SYSTEM TEST_BUTTON_LGHT (* System Configuration *)
  (* Standard: 61499-1 *)
  (* Version 0.3, 2003-12-05, JHC, Rockwell Automation, Renamed from NEWSYSTEM. *)
  (* Version 0.2, 2002-11-05, JHC, Rockwell Automation, Fixed missing (empty) FBD in Application. *)
  (* Version 0.1, 2002-01-17, JHC, Rockwell Automation, Minor cleanup *)
  (* Version 0.0, 2000-05-27, JHC, Rockwell Automation *)
  APPLICATION APP1
  END_APPLICATION
  DEVICE DEV1 : FRAME_DEVICE(BOUNDS := [100,100,100,100], GRID := [0,0])
    RESOURCE RES1 : PANEL_RESOURCE
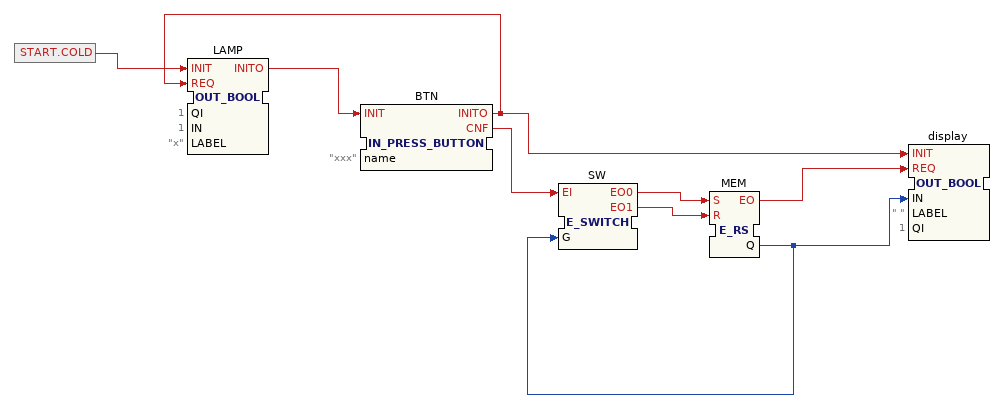
      FBS
        LAMP : OUT_BOOL(QI := 1, IN := 1, LABEL := "x");
        MEM : E_RS;
        BTN : IN_PRESS_BUTTON(name := "xxx");
        display : OUT_BOOL(LABEL := " ", QI := 1);
        SW : E_SWITCH;
      END_FBS
      EVENT_CONNECTIONS
        LAMP.INITO TO BTN.INIT;
        START.COLD TO LAMP.INIT;
        BTN.INITO TO LAMP.REQ;
        BTN.INITO TO display.INIT;
        MEM.EO TO display.REQ;
        SW.EO0 TO MEM.S;
        BTN.CNF TO SW.EI;
        SW.EO1 TO MEM.R;
      END_CONNECTIONS
      DATA_CONNECTIONS
        MEM.Q TO display.IN;
        MEM.Q TO SW.G;
      END_CONNECTIONS
    END_RESOURCE
  END_DEVICE
END_SYSTEM
